ABB RAPID module: Module1.mod

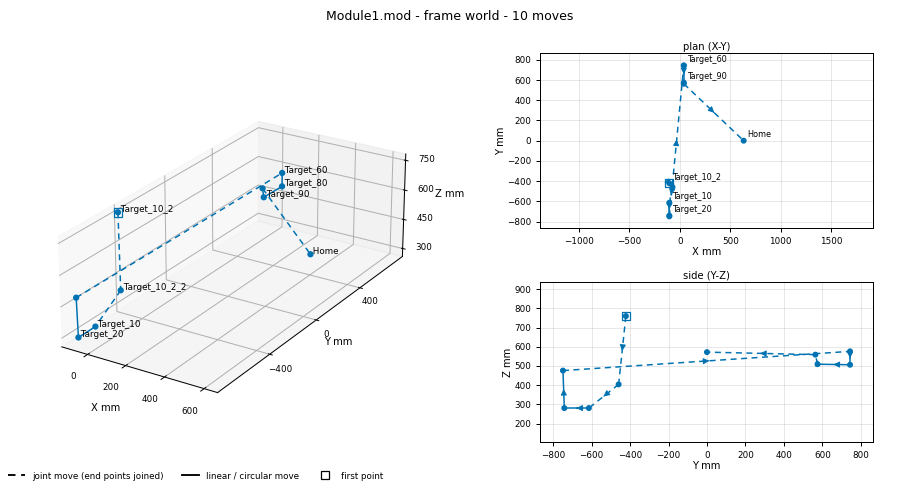
[picture p0: tool path of Module1.mod in frame world, 10 of 10 moves have a stored position in this frame; points joined in program order, loops and branches not executed]
MODULE Module1
        CONST robtarget Target_20:=[[-103.187,-742.033954446,281],[0.706105152,0.706105152,0.037623317,-0.037623317],[-1,-1,-2,6],[9E+09,9E+09,9E+09,9E+09,9E+09,9E+09]];
    CONST robtarget Target_10:=[[-103.187,-614.270973412,281],[0.706105152,0.706105152,0.037623317,-0.037623317],[-1,-1,-2,6],[9E+09,9E+09,9E+09,9E+09,9E+09,9E+09]];
    CONST robtarget Target_20_2:=[[-103.187,-748.994,476],[0.706105152,0.706105152,0.037623317,-0.037623317],[-1,-1,-2,6],[9E+09,9E+09,9E+09,9E+09,9E+09,9E+09]];
    CONST robtarget Target_40:=[[-98.1,645.70448909,536.344],[0.502606385,0.502606385,-0.497379957,-0.497379957],[1,-2,1,0],[9E+09,9E+09,9E+09,9E+09,9E+09,9E+09]];
    CONST robtarget Target_30:=[[-98.1,645.70448909,449.344],[0,0,0.707106781,0.707106781],[1,-2,1,0],[9E+09,9E+09,9E+09,9E+09,9E+09,9E+09]];
    CONST robtarget Target_50:=[[-98.1,502.323094749,449.344],[0,0,0.707106781,0.707106781],[1,-2,1,0],[9E+09,9E+09,9E+09,9E+09,9E+09,9E+09]];
    CONST robtarget Target_60:=[[39.815,744.179,576],[0.037623317,-0.037623317,0.706105152,0.706105152],[-2,-1,-2,6],[9E+09,9E+09,9E+09,9E+09,9E+09,9E+09]];
    CONST robtarget Target_20_2_2:=[[246.977782782,416.580570163,516],[0.182281552,0.182281552,-0.683208194,-0.683208194],[1,2,-3,0],[9E+09,9E+09,9E+09,9E+09,9E+09,9E+09]];
    CONST robtarget Target_20_2_3:=[[331.925997582,511.449773241,516],[0.207838237,0.207838237,-0.675872227,-0.675872227],[1,-2,1,0],[9E+09,9E+09,9E+09,9E+09,9E+09,9E+09]];
    CONST robtarget Target_90:=[[39.815,575.12025884,509.259598205],[0.037293563,-0.037950205,0.712240118,0.699916414],[-2,-1,-2,6],[9E+09,9E+09,9E+09,9E+09,9E+09,9E+09]];
    CONST robtarget Target_70:=[[39.815,634.823776433,516],[0,0,0.707106781,0.707106781],[-2,-1,-2,6],[9E+09,9E+09,9E+09,9E+09,9E+09,9E+09]];
    CONST robtarget Target_80:=[[39.815,744.179,506.304],[0.037293563,-0.037950205,0.712240118,0.699916414],[-2,-1,-2,6],[9E+09,9E+09,9E+09,9E+09,9E+09,9E+09]];
    CONST robtarget Home:=[[632.453792063,0,572.019237886],[0.353553391,0.612372436,0.612372436,0.353553391],[0,0,0,0],[9E+09,9E+09,9E+09,9E+09,9E+09,9E+09]];
    CONST robtarget Target_10_2:=[[-103.187,-421.828235204,759.553057669],[0.706105152,0.706105152,0.037623317,-0.037623317],[-1,-2,-1,6],[9E+09,9E+09,9E+09,9E+09,9E+09,9E+09]];
    CONST robtarget Target_10_2_2:=[[-71.646817737,-459.465576118,404.14050871],[0.706105152,0.706105152,0.037623317,-0.037623317],[-1,-1,-2,6],[9E+09,9E+09,9E+09,9E+09,9E+09,9E+09]];
    CONST robtarget Target_90_2:=[[39.815,563.87,558.804],[0.037623317,-0.037623317,0.706105152,0.706105152],[-2,-1,-2,6],[9E+09,9E+09,9E+09,9E+09,9E+09,9E+09]];
    CONST robtarget Target_100:=[[19.699463437,488.106384969,732.454156407],[0.012913401,0.015490597,0.76795361,0.640187893],[0,-1,0,0],[9E+09,9E+09,9E+09,9E+09,9E+09,9E+09]];
!***********************************************************
    !
    ! Module:  Module1
    !
    ! Description:
    !   <Insert description here>
    !
    ! Author: jecer
    !
    ! Version: 1.0
    !
    !***********************************************************


    !***********************************************************
    !
    ! Procedure main
    !
    !   This is the entry point of your program
    !
    !***********************************************************
    PROC main()
        WHILE TRUE DO
            Path_10;
        ENDWHILE
    ENDPROC
    PROC Path_10()
        WaitDI DI10_9,1;
        MoveJ Target_10_2,v400,z200,TCP1\WObj:=wobj0;
        MoveJ Target_10_2_2,v100,z200,TCP1\WObj:=wobj0;
        MoveJ Target_10,v100,fine,TCP1\WObj:=wobj0;
        MoveL Target_20,v60,fine,TCP1\WObj:=wobj0;
        WaitTime 0.5;
        MoveL Target_20_2,v60,z200,TCP1\WObj:=wobj0;
        MoveJ Target_60,v100,z100,TCP1\WObj:=Banda;
        MoveL Target_80,v20,fine,TCP1\WObj:=Banda;
        WaitTime 0.5;
        MoveL Target_90,v20,fine,TCP1\WObj:=Banda;
        MoveJ Target_90_2,v100,z200,TCP1\WObj:=Banda;
        PulseDO DO10_9;
        MoveJ Home,v400,z100,TCP1\WObj:=wobj0;
    ENDPROC
    PROC Path_20()
    ENDPROC
ENDMODULE
